{attribute 'qualified_only'}
{attribute 'strict'}
TYPE eAOTarget:
(
	manual 	:= 0,
	Genset	:= 1,
	hPU		:= 2
);
END_TYPE

(* stored: Version 1.1.0.1, ProductVersion 3.1.4026.18
   DUT eAOTarget: Id {3ec083b2-8f00-46d7-8417-fee2a168b131} *)
